FUNCTION_BLOCK CALIBRATE (* Two-point calibration (offset & scale) of an analog input with BOOL-triggered calibration. *)
  (* Standard: 61499-1; Description: version 1.3	11. mar. 2009 programmer 	hugo tested BY		hans *)
  (* Version 2.0, 2026-06-01, Meisterschulen am Ostbahnhof *)
  PACKAGE OSCAT::Basic::POUs::Engineering::measurements;
  (* Documentation:
  Formula
    Y = (X + OFFSET) * SCALE Calibration (Two-Point)
    - Offset (CO): Apply low reference, set Y_Offset to desired output, set CO=TRUE
   OFFSET := Y_Offset - X → shifts X so that Y = Y_Offset at this point
   - Scale (CS): Apply high reference, set Y_Scale to desired output, set CS=TRUE
   SCALE := Y_Scale / (X + OFFSET) → scales so that Y = Y_Scale at this point
    Note: Both Y_Offset and Y_Scale are target values on the output side.
   ⚠ IMPORTANT: CO must be executed before CS, because CS uses OFFSET from CO.
   In a SimpleFB this order cannot be enforced by the FB itself.
   See E_CALIBRATE_SQ for an event-driven variant with ECC-enforced sequencing.
   Example
   Scenario: 4–20 mA pressure sensor via logiBUS (0–10 V, normalized to 0.0..1.0).
   Desired output range: 0.0..500.0
      Step |  Action |  Result |  
    1 |  Apply 4 mA (X=0.0), set Y_Offset=0.0, CO=TRUE |  OFFSET = 0 |  
    2 |  Apply 20 mA (X=1.0), set Y_Scale=500.0, CS=TRUE |  SCALE = 500 |  
     Output: Y = (X + 0) * 500 = X * 500 = 0..500 ✓
  *)
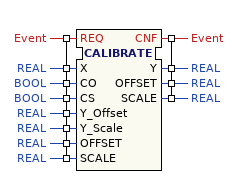
  EVENT_INPUT
    REQ WITH X, CO, CS, Y_Offset, Y_Scale, OFFSET, SCALE; (* Normal Execution Request *)
  END_EVENT
  EVENT_OUTPUT
    CNF WITH Y, OFFSET, SCALE; (* Execution Confirmation *)
  END_EVENT
  VAR_INPUT
    X : REAL; (* Input *)
    CO : BOOL; (* Calibrate Offset *)
    CS : BOOL; (* Calibrate Scale *)
    Y_Offset : REAL; (* Reference for offset calibration *)
    Y_Scale : REAL; (* Reference for scale calibration *)
  END_VAR
  VAR_OUTPUT
    Y : REAL; (* Calibrated Output *)
  END_VAR
  VAR_IN_OUT
    OFFSET : REAL := 0.0; (* Offset value *)
    SCALE : REAL := 1.0; (* Scale value *)
  END_VAR
  EC_STATES
    REQ : REQ -> CNF;
  END_STATES
  ALGORITHM REQ IN ST:
(* offset calibration: store offset so Y = Y_Offset at current X *)
IF CO THEN
	OFFSET := Y_Offset - X;
ELSIF CS THEN
	(* scale calibration: store scale so Y = Y_Scale at current X (requires OFFSET from CO!) *)
	IF (X + OFFSET) <> 0.0 THEN
		SCALE := Y_Scale / (X + OFFSET);
	END_IF;
END_IF;
(* calculate calibrated output *)
Y := (X + OFFSET) * SCALE;
  END_ALGORITHM
END_FUNCTION_BLOCK
